{attribute 'qualified_only'}
VAR_GLOBAL CONSTANT
	MAX_ITERABLE_ITEMS : INT := 20;
END_VAR

(* stored: Version 1.1.0.1, ProductVersion 3.1.4024.12
   GVL Param: Id {49f545d5-17b0-4af8-862d-44b9479f2ec7}, ParameterList True *)
